//{{V2}}
DATA_BLOCK DB1

AUTHOR:nb
FAMILY:nb
NAME:nb
VERSION:1.0


FB10

BEGIN

       Pulse:=FALSE
       Bit0:=FALSE
       Bit1:=FALSE
       Bit2:=FALSE
       int_val:=0
       fm:=FALSE
END_DATA_BLOCK
